{attribute 'linkalways'} 
{attribute 'no_explicit_call' := 'This FB is a CLASS and must be accessed using methods or properties'}
{attribute 'enable_dynamic_creation'}
FUNCTION_BLOCK _GVSP_IMAGE_INFO EXTENDS StructuredDatatypeBase
VAR
	localData : GVSP_IMAGE_INFO;
	activeData : REFERENCE TO GVSP_IMAGE_INFO REF= localData;
    _CameraIpAddress : _UDINT(localdata.CameraIpAddress);
    _LocalIpAddress : _UDINT(localdata.LocalIpAddress);
    _CameraUdpPort : _UINT(localdata.CameraUdpPort);
    _LocalUdpPort : _UINT(localdata.LocalUdpPort);
    _GvspChannelId : _UINT(localdata.GvspChannelId);
    _GevStatus : _UINT(localdata.GevStatus);
    _BlockId : _ULINT(localdata.BlockId);
    _LeaderInfo : _GVSP_LEADER_PAYLOAD_IMAGE();
END_VAR

PROPERTY PUBLIC Address : PVOID
GET
Address := ADR(activeData);
END_GET
END_PROPERTY

PROPERTY PUBLIC BlockId : REFERENCE TO _ULINT
GET
BlockId REF= _BlockId;
END_GET
END_PROPERTY

PROPERTY PUBLIC CameraIpAddress : REFERENCE TO _UDINT
GET
CameraIpAddress REF= _CameraIpAddress;
END_GET
END_PROPERTY

PROPERTY PUBLIC CameraUdpPort : REFERENCE TO _UINT
GET
CameraUdpPort REF= _CameraUdpPort;
END_GET
END_PROPERTY

METHOD PUBLIC ClearReference
VAR_INPUT
END_VAR
activeData REF= localData;
SetMemberReference();
END_METHOD

METHOD PUBLIC Clone : I_Datatype
VAR
    pClone : POINTER TO _GVSP_IMAGE_INFO;
END_VAR
pClone := __NEW(_GVSP_IMAGE_INFO());
pClone^.Value := Value;
Clone := pClone^;
END_METHOD

METHOD FB_init : BOOL
VAR_INPUT
	bInitRetains : BOOL; // if TRUE, the retain variables are initialized (warm start / cold start)
	bInCopyCode : BOOL;  // if TRUE, the instance afterwards gets moved into the copy code (online change)
END_VAR
SetMemberReference();
AddMember('CameraIpAddress', _CameraIpAddress);
AddMember('LocalIpAddress', _LocalIpAddress);
AddMember('CameraUdpPort', _CameraUdpPort);
AddMember('LocalUdpPort', _LocalUdpPort);
AddMember('GvspChannelId', _GvspChannelId);
AddMember('GevStatus', _GevStatus);
AddMember('BlockId', _BlockId);
AddMember('LeaderInfo', _LeaderInfo);
END_METHOD

PROPERTY PUBLIC GevStatus : REFERENCE TO _UINT
GET
GevStatus REF= _GevStatus;
END_GET
END_PROPERTY

PROPERTY PUBLIC GvspChannelId : REFERENCE TO _UINT
GET
GvspChannelId REF= _GvspChannelId;
END_GET
END_PROPERTY

PROPERTY PUBLIC Identifier : T_MAXSTRING
GET
Identifier := 'GVSP_IMAGE_INFO';
END_GET
END_PROPERTY

PROPERTY PUBLIC LeaderInfo : REFERENCE TO _GVSP_LEADER_PAYLOAD_IMAGE
GET
LeaderInfo REF= _LeaderInfo;
END_GET
END_PROPERTY

PROPERTY PUBLIC LocalIpAddress : REFERENCE TO _UDINT
GET
LocalIpAddress REF= _LocalIpAddress;
END_GET
END_PROPERTY

PROPERTY PUBLIC LocalUdpPort : REFERENCE TO _UINT
GET
LocalUdpPort REF= _LocalUdpPort;
END_GET
END_PROPERTY

METHOD PUBLIC MakeReferenceTo
VAR_INPUT
	ReferenceTarget : REFERENCE TO GVSP_IMAGE_INFO;
END_VAR
activeData REF= ReferenceTarget;
SetMemberReference();
END_METHOD

METHOD PROTECTED SetMemberReference
VAR_INPUT
END_VAR
_CameraIpAddress.MakeReferenceTo(activeData.CameraIpAddress);
_LocalIpAddress.MakeReferenceTo(activeData.LocalIpAddress);
_CameraUdpPort.MakeReferenceTo(activeData.CameraUdpPort);
_LocalUdpPort.MakeReferenceTo(activeData.LocalUdpPort);
_GvspChannelId.MakeReferenceTo(activeData.GvspChannelId);
_GevStatus.MakeReferenceTo(activeData.GevStatus);
_BlockId.MakeReferenceTo(activeData.BlockId);
_LeaderInfo.MakeReferenceTo(activeData.LeaderInfo);
END_METHOD

PROPERTY PUBLIC Size : UDINT
GET
Size := SIZEOF(activeData);
END_GET
END_PROPERTY

METHOD TryMakeReferenceTo : BOOL
VAR_INPUT
	Target : I_Datatype;
END_VAR
VAR
	targetAsStruct : I_StructuredDatatype;
	pTargetData : POINTER TO GVSP_IMAGE_INFO;
END_VAR
IF NOT Target.TryResolveAsStructuredDatatype(targetAsStruct) THEN
	RETURN;
END_IF

IF NOT (targetAsStruct.Identifier = Identifier) THEN
	RETURN;
END_IF

pTargetData := Target.Address;
activeData REF= pTargetData^;
SetMemberReference();
TryMakeReferenceTo := TRUE;
END_METHOD

PROPERTY PUBLIC Value : REFERENCE TO GVSP_IMAGE_INFO
GET
Value REF= activeData;
END_GET
END_PROPERTY

END_FUNCTION_BLOCK

(* stored: Version 1.1.0.1, ProductVersion 3.1.4024.13
   POU _GVSP_IMAGE_INFO: Id {da5781c1-fb67-05f6-2284-0e8262f9113b}, SpecialFunc None
   Folder Core: Id {5f39f996-c21b-05d4-18a8-6a1cfd531274}
   Folder Customize: Id {774670f1-3574-0e96-156c-c57156ffae8e}
   Folder Constructor: Id {e41327a1-1298-0a7b-3eae-19c74fae01cb}
   Folder Protected: Id {f2758d70-fd82-0cc5-2823-6d23786424c0}
   Property Address: Id {71fb01c0-8396-0eab-36cd-bed8e4be6688}
   Get Get: Id {6df94c81-a2bc-0306-2713-6da57b816928}
   Property BlockId: Id {1d9e0593-53c3-0087-16b3-f15f74162e41}
   Get Get: Id {a61be0e6-69d7-0479-1609-8fbd1e631a83}
   Property CameraIpAddress: Id {bdd9e853-49ba-022b-2cda-98b485890295}
   Get Get: Id {de9af7cc-27c4-02d5-15b1-8339aa0f928d}
   Property CameraUdpPort: Id {325ea0fd-949d-0ff7-1d5f-b16dd05f36af}
   Get Get: Id {a8bb9db8-144e-03da-00ad-a7f54924fbe7}
   Method ClearReference: Id {aaa9697f-df45-0ef7-12e4-b51a41fa131e}
   Method Clone: Id {ca3defd2-62f7-0ccc-14e6-4eefd2e01ed8}
   Method FB_init: Id {41e44d81-40bb-05c3-0a99-7c7152efbd3c}
   Property GevStatus: Id {dda42ad0-c5bb-0978-3190-16359d903a07}
   Get Get: Id {136df57b-1818-01ff-0179-2d7491d6ba5b}
   Property GvspChannelId: Id {cf365d6a-e546-0b3d-080c-766768ff1ae3}
   Get Get: Id {6ed5047d-0890-09f3-1463-4a4ebb6ed70c}
   Property Identifier: Id {720a60b2-4bec-0c06-08bf-c0b07066ff55}
   Get Get: Id {aaec201b-cbcf-0a57-0809-0cb3ffe8ff82}
   Property LeaderInfo: Id {1fac3339-48b8-04f3-0c00-a587943d5c28}
   Get Get: Id {acd08174-9fac-0c2e-19a7-7e61b34de92e}
   Property LocalIpAddress: Id {36505468-3a8e-0a97-35cf-7ac5f4619047}
   Get Get: Id {89a716e4-0a79-0901-3fee-99f11ab750e6}
   Property LocalUdpPort: Id {986fd1af-1295-0557-3c4e-81b69e0d6a58}
   Get Get: Id {de66a537-33e4-0249-0c5e-367f3803ec4e}
   Method MakeReferenceTo: Id {22bd43e8-76e2-0f6c-0872-a59434bdba8d}
   Method SetMemberReference: Id {82879577-1d75-0c73-0985-2aa201a04948}
   Property Size: Id {ec6346e1-6e7d-03c8-27de-0d9270613808}
   Get Get: Id {faa4fa95-b697-0dcd-0d2b-a3af3eaf7a33}
   Method TryMakeReferenceTo: Id {e4c785bf-4d72-0fa9-2511-48a6f9970c59}
   Property Value: Id {fcdd44c8-ecf9-06c0-1a2a-0c1963747971}
   Get Get: Id {32c02205-1a3d-0bbe-21a8-f25f036ca8ea} *)
